// TIA Portal V20 export
// export: Created 2025-12-01T14:57:26.7593749Z, ExportSetting None, DisplayName Totally Integrated Automation Portal, DisplayVersion V20 Update 3, DisplayName TIA Portal Openness, DisplayVersion V20 Update 3, DisplayName TIA Portal Version Control Interface, DisplayVersion V20 Update 3, DisplayName STEP 7 Professional, DisplayVersion V20 Update 3, DisplayName STEP 7 Safety, DisplayVersion V20 Update 2, DisplayName WinCC Basic/Comfort/Advanced, DisplayVersion V20 Update 3, DisplayName WinCC Professional, DisplayVersion V20 Update 3, DisplayName WinCC Unified, DisplayVersion V20 Update 3
FUNCTION "FC604_PuntoBorradoDatos_Quimarox" : Void   // FC604, LAD
{ S7_Optimized_Access := 'FALSE' }
// stored: AutoNumber false, SetENOAutomatically false
   VAR_INPUT
      ID_Quimarox : Int;
      ID_Elemento : Int;
   END_VAR
   VAR_TEMP
      Nux_NumeroVagon : Int;
   END_VAR
BEGIN

NETWORK
TITLE = Borrar el Peine del Quimarox
//======================================================================================================================================
// sacamos el dato del vagón que tenemos en frente del elemento:
      L     "DB602_ElementosQuimarox".Quimarox[#ID_Quimarox].Elementos[#ID_Elemento].Numero_carrier;
      T     #Nux_NumeroVagon;

// Numero de Vagon nunca debe ser CERO
      L     #Nux_NumeroVagon;
      L     0;
      ==I;
      JC    fin;

// Hay Carrier en ventana
      SET;
      AN    "DB602_ElementosQuimarox".Quimarox[#ID_Quimarox].Elementos[#ID_Elemento].Hay_Carrier_en_ventana;
      JC    fin;

// primero comprobamos si tenemos algún mensaje pendiente de emitir
      SET;
      L     "DB601_PeinesQuimarox".Quimarox[#ID_Quimarox].vagon[#Nux_NumeroVagon].EventoAGenerar;
      L     0;
      <>I;
      JC    fin;


//========================================================================================================================================
// borramos los datos del vagón, salvo los de la reserva
      SET;
      R     "DB601_PeinesQuimarox".Quimarox[#ID_Quimarox].vagon[#Nux_NumeroVagon].Carrier_Cargado;
      R     "DB601_PeinesQuimarox".Quimarox[#ID_Quimarox].vagon[#Nux_NumeroVagon].vagon_cargado_SinDestino;
      R     "DB601_PeinesQuimarox".Quimarox[#ID_Quimarox].vagon[#Nux_NumeroVagon].carrier_multiple;
//      R     "DB601_DatosPeinesQuimarox".Quimarox[#ID_Quimarox].vagon[#Nux_NumeroVagon].vagon_reservado_carga

      L     0;
      T     "DB601_PeinesQuimarox".Quimarox[#ID_Quimarox].vagon[#Nux_NumeroVagon].Destino_principal;
      T     "DB601_PeinesQuimarox".Quimarox[#ID_Quimarox].vagon[#Nux_NumeroVagon].Destino_alternativo;
      T     "DB601_PeinesQuimarox".Quimarox[#ID_Quimarox].vagon[#Nux_NumeroVagon].Mesa_descarga;
      T     "DB601_PeinesQuimarox".Quimarox[#ID_Quimarox].vagon[#Nux_NumeroVagon].Num_Recirculaciones;
      T     "DB601_PeinesQuimarox".Quimarox[#ID_Quimarox].vagon[#Nux_NumeroVagon].Numero_Vagones_Multiple_Asociados;
//      T     "DB601_DatosPeinesQuimarox".Quimarox[#ID_Quimarox].vagon[#Nux_NumeroVagon].punto_entrada_carga

      L     0;
      T     "DB601_PeinesQuimarox".Quimarox[#ID_Quimarox].vagon[#Nux_NumeroVagon].EventoAGenerar;
      T     "DB601_PeinesQuimarox".Quimarox[#ID_Quimarox].vagon[#Nux_NumeroVagon].DatosCarga.Mckey;
      T     "DB601_PeinesQuimarox".Quimarox[#ID_Quimarox].vagon[#Nux_NumeroVagon].DatosCarga.MesaDestino;
      T     "DB601_PeinesQuimarox".Quimarox[#ID_Quimarox].vagon[#Nux_NumeroVagon].DatosCarga.MesaOrigen;
      T     "DB601_PeinesQuimarox".Quimarox[#ID_Quimarox].vagon[#Nux_NumeroVagon].DatosCarga.EtiquetaRouter;




//========================================================================================================================================
fin:  BE;
END_FUNCTION
